// TIA Portal V17 export
// export: Created 2024-09-15T12:30:30.8670403Z, ExportSetting WithDefaults, DisplayName Totally Integrated Automation Portal, DisplayVersion V17, DisplayName TIA Portal Openness, DisplayVersion V17, DisplayName TIA Portal Version Control Interface, DisplayVersion V17, DisplayName STEP 7 Professional, DisplayVersion V17, DisplayName STEP 7 Safety, DisplayVersion V17, DisplayName WinCC Professional, DisplayVersion V17
TYPE "typ_MQTT_ Interface_Dashboard_Publish"
// stored: IsFailsafeCompliant false
   STRUCT
      ldt_AcknowledgeButton : LDT;
      ConfigRateEnvironmentSensor : "typ_Config_Environment_Sensor";
      ConfigRateBrightnessSensor : "typ_Config_Brightness_Sensor";
      ConfigRateCameraPicture : "typ_Config_Camera_Picture";
      PosPanTiltUnit { S7_SetPoint := 'True'} : "typ_Pos_Pan_Tilt_Unit_Mov";
      OrderWorkpieceButton : "typ_Order_Workpiece_Buttons";
      ActionButtonNFCModule : "typ_Action_Buttons_NFC_Module";
   END_STRUCT;
END_TYPE
